// Mitsubishi GX Works2 project: pump_chem_up   PLC: FX3U/FX3UC

PROGRAM MAIN
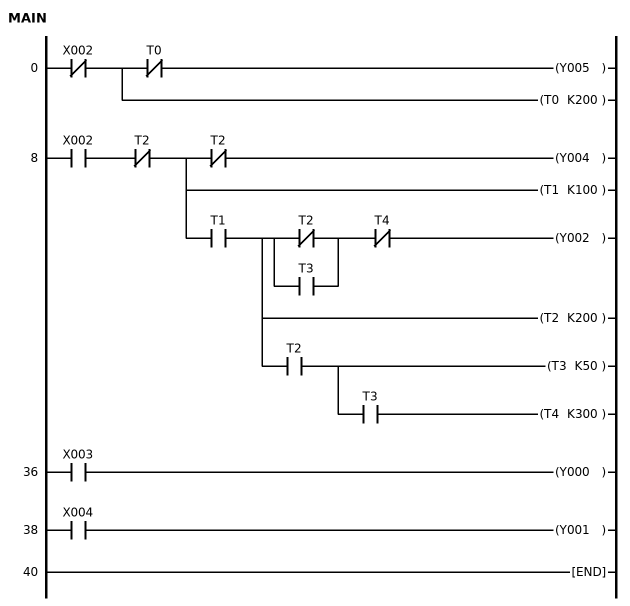
0     LDI     X002
      MPS
      ANI     T0
      OUT     Y005
      MPP
      OUT     T0 K200
8     LD      X002
      ANI     T2
      MPS
      ANI     T2
      OUT     Y004
      MPP
      OUT     T1 K100
      AND     T1
      MPS
      LDI     T2
      OR      T3
      ANB
      ANI     T4
      OUT     Y002
      MPP
      OUT     T2 K200
      AND     T2
      OUT     T3 K50
      AND     T3
      OUT     T4 K300
36    LD      X003
      OUT     Y000
38    LD      X004
      OUT     Y001
40    END
END_PROGRAM
